FUNCTION_BLOCK FB_AlarmResets
VAR_INPUT
END_VAR
VAR_OUTPUT
END_VAR
VAR
	//ACTION THIS SHOULD BE A PRPGRAM AND NOT A FUNCTION BLOCK. USING GLOBAL VARS

	ManualAlarmReset:	TP;			(* One second pulse for manual alarm reset *)
	AutomaticReset:	TP;			(*    One second pulse for automatic alarm reset, only in stop mode every e.g. 10 seconds *)
	AutomaticResetTiming: TON; 	(* Interval timer for automatic resets*)
	rtrigManualReset: R_TRIG;
	TPResetAfterGridFailure: TP;
	TONResetAfterGridFailure: TON;
	rtrigManualSafetyReset: R_TRIG;
	SafetyAlarmReset: TP;
END_VAR

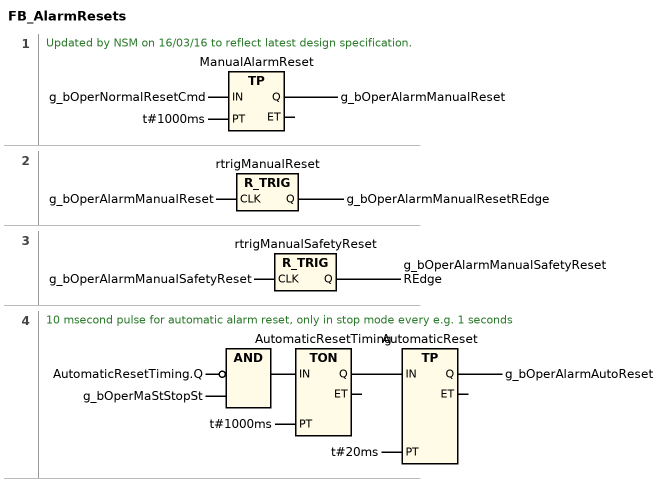
// NETWORK 1
// 					Updated by NSM on 16/03/16 to reflect latest design specification.
//
//
//
//
ManualAlarmReset(IN := g_bOperNormalResetCmd, PT := t#1000ms); // TP
g_bOperAlarmManualReset := ManualAlarmReset.Q;

// NETWORK 2
rtrigManualReset(CLK := g_bOperAlarmManualReset); // R_TRIG
g_bOperAlarmManualResetREdge := rtrigManualReset.Q;

// NETWORK 3
rtrigManualSafetyReset(CLK := g_bOperAlarmManualSafetyReset); // R_TRIG
g_bOperAlarmManualSafetyResetREdge := rtrigManualSafetyReset.Q;

// NETWORK 4
// 10 msecond pulse for automatic alarm reset, only in stop mode every e.g. 1 seconds
AutomaticResetTiming(IN := NOT AutomaticResetTiming.Q AND g_bOperMaStStopSt, PT := t#1000ms); // TON
AutomaticReset(IN := AutomaticResetTiming.Q, PT := t#20ms); // TP
g_bOperAlarmAutoReset := AutomaticReset.Q;

END_FUNCTION_BLOCK

(* stored: Version 1.1.0.1, ProductVersion 3.1.4024.9
   POU FB_AlarmResets: Id {ca0f5e23-d4ce-40f7-bc02-8dd9e65cf57b}, SpecialFunc None *)
